FUNCTION AI_OOR : BOOL
VAR_INPUT
	Status : WORD;
END_VAR

// calculate whether the status for an analog input is indicating an error
// the error bit is the 7th bit of the status word
// access to bits is base 0, so the 7th bit is accessed with index 6

AI_OOR := Status.6;

END_FUNCTION

(* stored: Version 1.1.0.1, ProductVersion 3.1.4024.12
   POU AI_OOR: Id {e625b465-b3a8-4c57-b528-1559e093f5e4}, SpecialFunc None *)
